// SIMATIC S7-200 project (STEP 7-Micro/WIN), CPU 226 REL 01.23

SYMBOL_TABLE USER1
start_button     I0.0     // start button
stop_button      I0.1     // stop button
inner_c_1_m      I0.2     // inner calling for first floor ( modern lift )
inner_c_2_m      I0.3     // inner calling for second floor ( modern lift )
inner_c_3_m      I0.4     // inner calling for third floor ( modern lift )
emergency_button I0.5     // system emergency button ( modern lift )
door_sensor_m    I0.6     // cabin door sensor ( modern lift )
bottom_limit_m   I0.7     // bottom limit sensor ( modern lift )
top_limit_m      I1.0     // top limit sensor ( modern lift )
floor_1_limit_m  I1.1     // first floor sensor ( modern lift )
floor_2_limit_m  I1.2     // second floor sensor ( modern lift )
floor_3_limit_m  I1.3     // third floor sensor ( modern lift )
floor_1_limit_o  I1.4     // first floor sensor ( old lift )
floor_2_limit_o  I1.5     // second floor sensor ( old lift )
floor_3_limit_o  I1.6     // third floor sensor ( old lift )
inner_c_1_o      I2.4     // inner calling for first floor ( old lift )
inner_c_2_o      I2.5     // inner calling for second floor ( old lift )
inner_c_3_o      I2.6     // inner calling for third floor ( old lift )
outer_c_1        I2.0     // outer calling for first floor
outer_c_2_d      I2.1     // outer calling for second floor in purpose of moving down
outer_c_2_u      I2.2     // outer calling for second floor in purpose of moving up
outer_c_3        I2.3     // outer calling for third floor
data_a_m         Q0.0     // data  a  for  (7447 7_segment) circuit  ( modern lift )
data_b_m         Q0.1     // data  b  for  (7447 7_segment) circuit  ( modern lift )
floor_1_led_m    Q0.2     // first floor calling led  ( modern lift )
floor_2_led_m    Q0.3     // second floor calling led  ( modern lift )
floor_3_led_m    Q0.4     // third floor calling led  ( modern lift )
emergency_led    Q0.5     // emergency calling led  ( modern lift )
door_lock_m      Q0.6     // security lock open/close output for lift cabin door  ( modern lift )
lighting_m       Q0.7     // cabin  inside lighting  ( modern lift )
cabin_down_m     Q1.0     // output for the lift motor for down movement  ( modern lift )
cabin_up_m       Q1.1     // output for the lift motor for up movement  ( modern lift )
cabin_down_o     Q1.3     // output for the lift motor for down movement  ( old lift )
cabin_up_o       Q1.2     // output for the lift motor for up movement  ( old lift )
functional_timer_off_1 T37      // functional_timer_off is used specially for inside cabin lighting
functional_timer_off_2 T38      // functional_timer_off is used in purpose of delaying between calls (modern lift)
functional_timer_off_3 T39      // functional_timer_off is used in purpose of delaying between calls (old lift)
functional_byte_1 VB0      // functional_byte_is used to determine in which floor is modern lift
functional_byte_2 VB1      // functional_byte_is used to determine in which floor is old lif
functional_bit_0 V6.0     // bit used for downloading the starting constraints in sbr(1) and sbr(2)
functional_bit_1 V6.1     // bit used for downloading the starting constraints in sbr(3)
functional_bit_2 V6.2     // bit used for downloading the starting constraints in sbr(4)
functional_bit_3 V6.3     // bit used for downloading the starting constraints in sbr(5)
functional_bit_4 V6.4     // bit used for downloading the starting constraints in sbr(6)
functional_bit_5 V6.5     // bit used for downloading the starting constraints in sbr(7)
functional_bit_6 V6.6     // bit used for downloading the starting constraints in sbr(11)
functional_bit_7 V6.7     // bit used for downloading the starting constraints in sbr(12)
functional_bit_8 V7.0     // bit used for downloading the starting constraints in sbr(13)
functional_bit_9 V7.1     // bit used for downloading the starting constraints in sbr(14)
system_on_off    M0.0     // system  on/off contact
sbr_1_call_bit   M0.1     // subroutine (1) calling bit
sbr_2_call_bit   M0.2     // subroutine (2) calling bit
sbr_3_call_bit   M0.3     // subroutine (3) calling bit
sbr_4_call_bit   M0.4     // subroutine (4) calling bit
sbr_5_call_bit   M0.5     // subroutine (5) calling bit
sbr_6_call_bit   M0.6     // subroutine (6) calling bit
sbr_7_call_bit   M0.7     // subroutine (7) calling bit
sbr_11_call_bit  M2.3     // subroutine (11) calling bit
sbr_12_call_bit  M2.7     // subroutine (12) calling bit
sbr_13_call_bit  M3.0     // subroutine (13) calling bit
sbr_14_call_bit  M3.1     // subroutine (14) calling bit
m_1_to_2         M1.0     // it is made set while modern lift is moving from floor 1 to floor 2
m_2_to_3         M1.1     // it is made set while modern lift is moving from floor 2 to floor 3
m_2_to_1         M1.2     // it is made set while modern lift is moving from floor 2 to floor 1
m_3_to_2         M1.3     // it is made set while modern lift is moving from floor 3 to floor 2
m_busy           M1.4     // it is made set while modern lift is busy
o_1_to_2         M1.5     // it is made set while old lift is moving from floor 1 to floor 2
o_2_to_3         M1.6     // it is made set while old lift is moving from floor 2 to floor 3
o_2_to_1         M1.7     // it is made set while old lift is moving from floor 2 to floor 1
o_3_to_2         M2.0     // it is made set while old lift is moving from floor 3 to floor 2
o_busy           M2.1     // it is made set while old lift is busy
both_ready       M2.2     // it is made set when both lifts are ready
m_busy_o_ready   M2.4     // it is made set when modren lift is busy and old lift is ready
m_ready_o_busy   M2.5     // it is made set when modren lift is ready and old lift is busy
both_busy        M2.6     // it is made set when both lifts are busy
First_Scan_On    SM0.1    // ON for the first scan cycle only
Always_On        SM0.0    // Always ON
END_SYMBOL_TABLE

ORGANIZATION_BLOCK MAIN:OB1
TITLE=control two lifts (modern and old) to work in priority
BEGIN
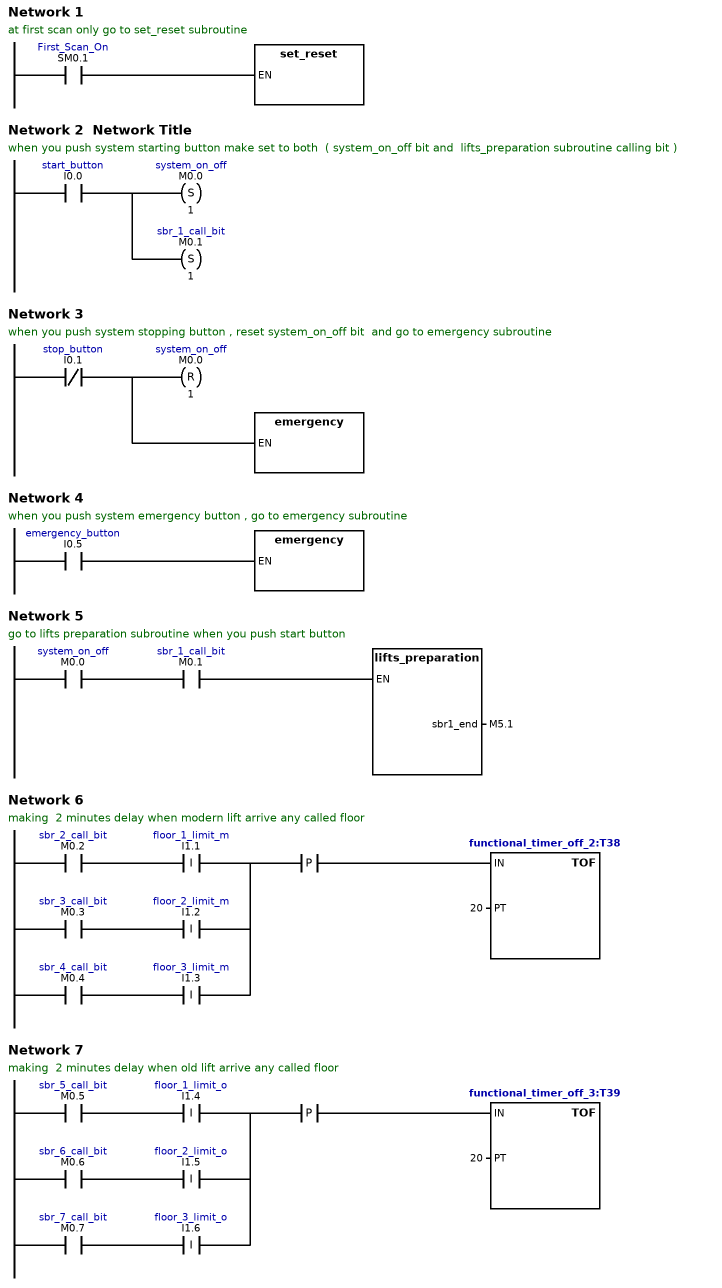
Network 1
// at first scan only go to set_reset subroutine
LD     First_Scan_On:SM0.1
CALL   set_reset:SBR0
Network 2 // Network Title
// when you push system starting button make set to both  ( system_on_off bit and  lifts_preparation subroutine calling bit )
LD     start_button:I0.0
S      system_on_off:M0.0, 1
S      sbr_1_call_bit:M0.1, 1
Network 3
// when you push system stopping button , reset system_on_off bit  and go to emergency subroutine
LDN    stop_button:I0.1
R      system_on_off:M0.0, 1
CALL   emergency:SBR15
Network 4
// when you push system emergency button , go to emergency subroutine
LD     emergency_button:I0.5
CALL   emergency:SBR15
Network 5
// go to lifts preparation subroutine when you push start button
LD     system_on_off:M0.0
A      sbr_1_call_bit:M0.1
CALL   lifts_preparation:SBR1, M5.1
Network 6
// making  2 minutes delay when modern lift arrive any called floor
LD     sbr_2_call_bit:M0.2
AI     floor_1_limit_m:I1.1
LD     sbr_3_call_bit:M0.3
AI     floor_2_limit_m:I1.2
OLD
LD     sbr_4_call_bit:M0.4
AI     floor_3_limit_m:I1.3
OLD
EU
TOF    functional_timer_off_2:T38, 20
Network 7
// making  2 minutes delay when old lift arrive any called floor
LD     sbr_5_call_bit:M0.5
AI     floor_1_limit_o:I1.4
LD     sbr_6_call_bit:M0.6
AI     floor_2_limit_o:I1.5
OLD
LD     sbr_7_call_bit:M0.7
AI     floor_3_limit_o:I1.6
OLD
EU
TOF    functional_timer_off_3:T39, 20
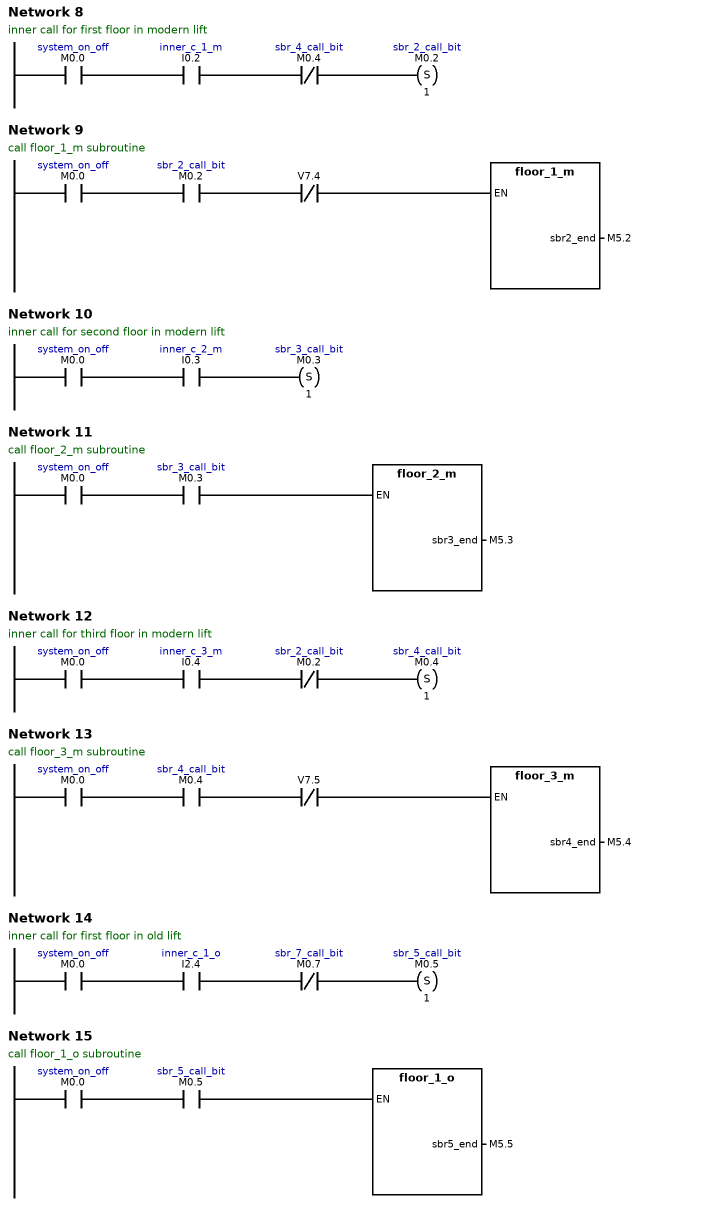
Network 8
// inner call for first floor in modern lift
LD     system_on_off:M0.0
A      inner_c_1_m:I0.2
AN     sbr_4_call_bit:M0.4
S      sbr_2_call_bit:M0.2, 1
Network 9
// call floor_1_m subroutine
LD     system_on_off:M0.0
A      sbr_2_call_bit:M0.2
AN     V7.4
CALL   floor_1_m:SBR2, M5.2
Network 10
// inner call for second floor in modern lift
LD     system_on_off:M0.0
A      inner_c_2_m:I0.3
S      sbr_3_call_bit:M0.3, 1
Network 11
// call floor_2_m subroutine
LD     system_on_off:M0.0
A      sbr_3_call_bit:M0.3
CALL   floor_2_m:SBR3, M5.3
Network 12
// inner call for third floor in modern lift
LD     system_on_off:M0.0
A      inner_c_3_m:I0.4
AN     sbr_2_call_bit:M0.2
S      sbr_4_call_bit:M0.4, 1
Network 13
// call floor_3_m subroutine
LD     system_on_off:M0.0
A      sbr_4_call_bit:M0.4
AN     V7.5
CALL   floor_3_m:SBR4, M5.4
Network 14
// inner call for first floor in old lift
LD     system_on_off:M0.0
A      inner_c_1_o:I2.4
AN     sbr_7_call_bit:M0.7
S      sbr_5_call_bit:M0.5, 1
Network 15
// call floor_1_o subroutine
LD     system_on_off:M0.0
A      sbr_5_call_bit:M0.5
CALL   floor_1_o:SBR5, M5.5
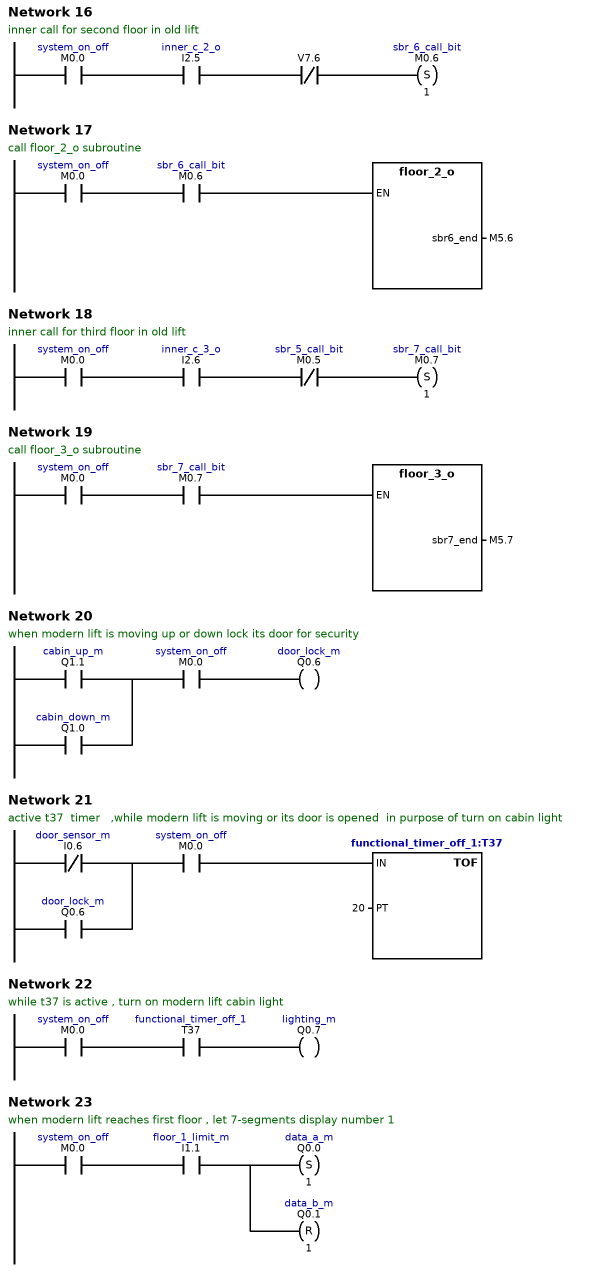
Network 16
// inner call for second floor in old lift
LD     system_on_off:M0.0
A      inner_c_2_o:I2.5
AN     V7.6
S      sbr_6_call_bit:M0.6, 1
Network 17
// call floor_2_o subroutine
LD     system_on_off:M0.0
A      sbr_6_call_bit:M0.6
CALL   floor_2_o:SBR6, M5.6
Network 18
// inner call for third floor in old lift
LD     system_on_off:M0.0
A      inner_c_3_o:I2.6
AN     sbr_5_call_bit:M0.5
S      sbr_7_call_bit:M0.7, 1
Network 19
// call floor_3_o subroutine
LD     system_on_off:M0.0
A      sbr_7_call_bit:M0.7
CALL   floor_3_o:SBR7, M5.7
Network 20
// when modern lift is moving up or down lock its door for security
LD     cabin_up_m:Q1.1
O      cabin_down_m:Q1.0
A      system_on_off:M0.0
=      door_lock_m:Q0.6
Network 21
// active t37  timer   ,while modern lift is moving or its door is opened  in purpose of turn on cabin light
LDN    door_sensor_m:I0.6
O      door_lock_m:Q0.6
A      system_on_off:M0.0
TOF    functional_timer_off_1:T37, 20
Network 22
// while t37 is active , turn on modern lift cabin light 
LD     system_on_off:M0.0
A      functional_timer_off_1:T37
=      lighting_m:Q0.7
Network 23
// when modern lift reaches first floor , let 7-segments display number 1
LD     system_on_off:M0.0
A      floor_1_limit_m:I1.1
S      data_a_m:Q0.0, 1
R      data_b_m:Q0.1, 1
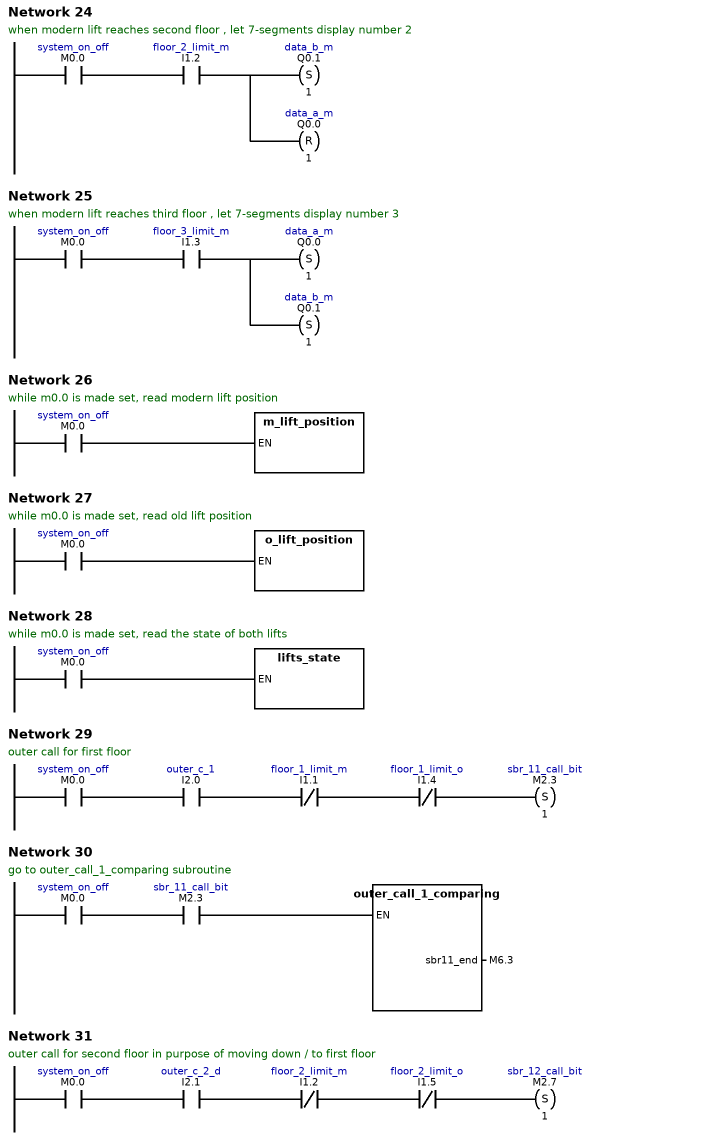
Network 24
// when modern lift reaches second floor , let 7-segments display number 2
LD     system_on_off:M0.0
A      floor_2_limit_m:I1.2
S      data_b_m:Q0.1, 1
R      data_a_m:Q0.0, 1
Network 25
// when modern lift reaches third floor , let 7-segments display number 3
LD     system_on_off:M0.0
A      floor_3_limit_m:I1.3
S      data_a_m:Q0.0, 1
S      data_b_m:Q0.1, 1
Network 26
// while m0.0 is made set, read modern lift position
LD     system_on_off:M0.0
CALL   m_lift_position:SBR8
Network 27
// while m0.0 is made set, read old lift position
LD     system_on_off:M0.0
CALL   o_lift_position:SBR9
Network 28
// while m0.0 is made set, read the state of both lifts
LD     system_on_off:M0.0
CALL   lifts_state:SBR10
Network 29
// outer call for first floor  
LD     system_on_off:M0.0
A      outer_c_1:I2.0
AN     floor_1_limit_m:I1.1
AN     floor_1_limit_o:I1.4
S      sbr_11_call_bit:M2.3, 1
Network 30
// go to outer_call_1_comparing subroutine
LD     system_on_off:M0.0
A      sbr_11_call_bit:M2.3
CALL   outer_call_1_comparing:SBR11, M6.3
Network 31
// outer call for second floor in purpose of moving down / to first floor
LD     system_on_off:M0.0
A      outer_c_2_d:I2.1
AN     floor_2_limit_m:I1.2
AN     floor_2_limit_o:I1.5
S      sbr_12_call_bit:M2.7, 1
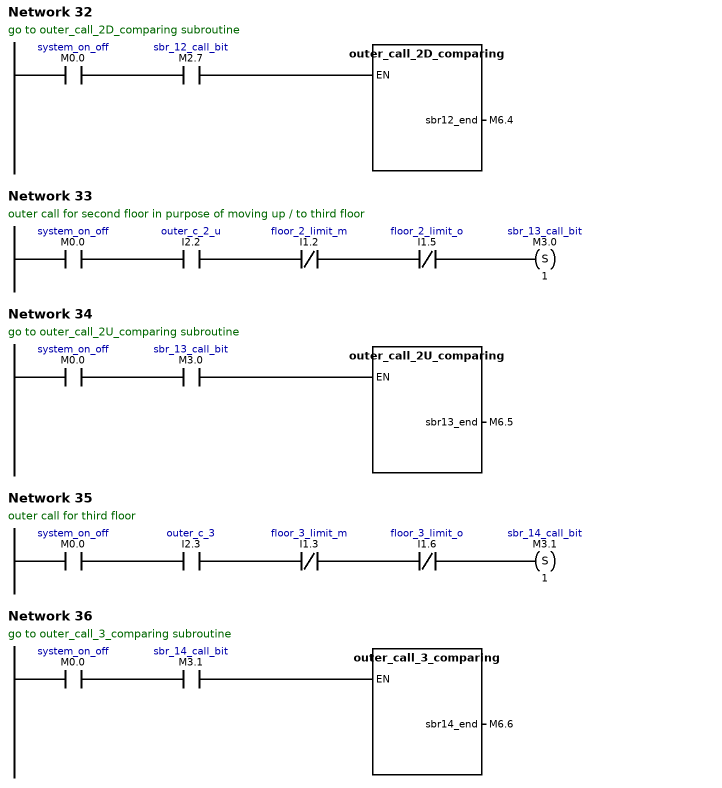
Network 32
// go to outer_call_2D_comparing subroutine
LD     system_on_off:M0.0
A      sbr_12_call_bit:M2.7
CALL   outer_call_2D_comparing:SBR12, M6.4
Network 33
// outer call for second floor in purpose of moving up / to third floor
LD     system_on_off:M0.0
A      outer_c_2_u:I2.2
AN     floor_2_limit_m:I1.2
AN     floor_2_limit_o:I1.5
S      sbr_13_call_bit:M3.0, 1
Network 34
// go to outer_call_2U_comparing subroutine
LD     system_on_off:M0.0
A      sbr_13_call_bit:M3.0
CALL   outer_call_2U_comparing:SBR13, M6.5
Network 35
// outer call for third floor 
LD     system_on_off:M0.0
A      outer_c_3:I2.3
AN     floor_3_limit_m:I1.3
AN     floor_3_limit_o:I1.6
S      sbr_14_call_bit:M3.1, 1
Network 36
// go to outer_call_3_comparing subroutine
LD     system_on_off:M0.0
A      sbr_14_call_bit:M3.1
CALL   outer_call_3_comparing:SBR14, M6.6
END_ORGANIZATION_BLOCK

SUBROUTINE_BLOCK set_reset:SBR0
TITLE=put all memories , timers and outputs that are used in program at initial position 
BEGIN
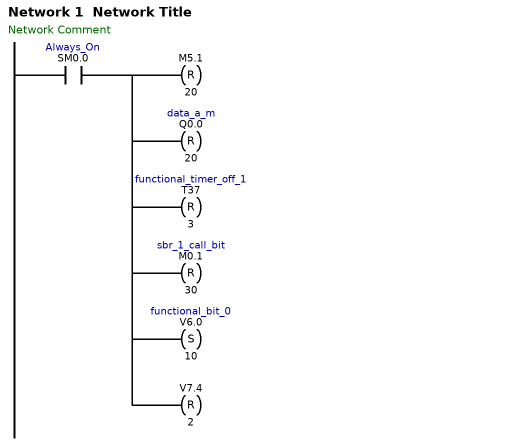
Network 1 // Network Title
// Network Comment
LD     Always_On:SM0.0
R      M5.1, 20
R      data_a_m:Q0.0, 20
R      functional_timer_off_1:T37, 3
R      sbr_1_call_bit:M0.1, 30
S      functional_bit_0:V6.0, 10
R      V7.4, 2
END_SUBROUTINE_BLOCK

SUBROUTINE_BLOCK lifts_preparation:SBR1
TITLE=move modern lift to third floor and old lift to first floor 
VAR_OUTPUT
sbr1_end:BOOL;	// L0.0 
END_VAR
BEGIN
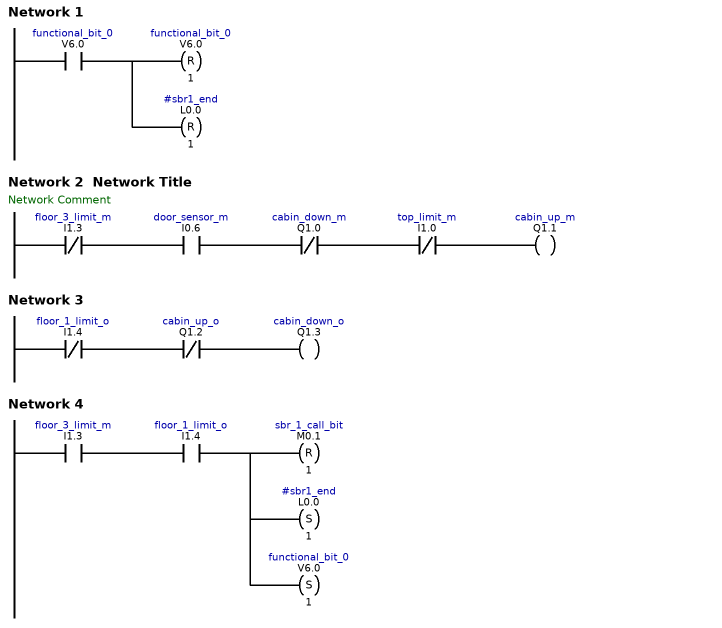
Network 1
LD     functional_bit_0:V6.0
R      functional_bit_0:V6.0, 1
R      #sbr1_end:L0.0, 1
Network 2 // Network Title
// Network Comment
LDN    floor_3_limit_m:I1.3
A      door_sensor_m:I0.6
AN     cabin_down_m:Q1.0
AN     top_limit_m:I1.0
=      cabin_up_m:Q1.1
Network 3
LDN    floor_1_limit_o:I1.4
AN     cabin_up_o:Q1.2
=      cabin_down_o:Q1.3
Network 4
LD     floor_3_limit_m:I1.3
A      floor_1_limit_o:I1.4
R      sbr_1_call_bit:M0.1, 1
S      #sbr1_end:L0.0, 1
S      functional_bit_0:V6.0, 1
END_SUBROUTINE_BLOCK

SUBROUTINE_BLOCK floor_1_m:SBR2
TITLE=move modern lift to first floor
VAR_OUTPUT
sbr2_end:BOOL;	// L0.0 
END_VAR
BEGIN
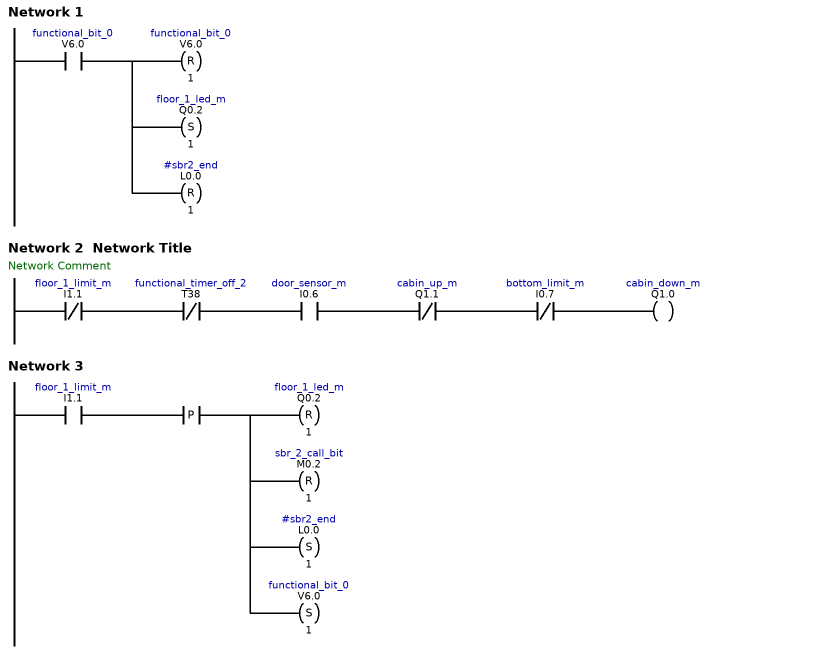
Network 1
LD     functional_bit_0:V6.0
R      functional_bit_0:V6.0, 1
S      floor_1_led_m:Q0.2, 1
R      #sbr2_end:L0.0, 1
Network 2 // Network Title
// Network Comment
LDN    floor_1_limit_m:I1.1
AN     functional_timer_off_2:T38
A      door_sensor_m:I0.6
AN     cabin_up_m:Q1.1
AN     bottom_limit_m:I0.7
=      cabin_down_m:Q1.0
Network 3
LD     floor_1_limit_m:I1.1
EU
R      floor_1_led_m:Q0.2, 1
R      sbr_2_call_bit:M0.2, 1
S      #sbr2_end:L0.0, 1
S      functional_bit_0:V6.0, 1
END_SUBROUTINE_BLOCK

SUBROUTINE_BLOCK floor_2_m:SBR3
TITLE=move modern lift to second floor
VAR_OUTPUT
sbr3_end:BOOL;	// L0.0 
END_VAR
BEGIN
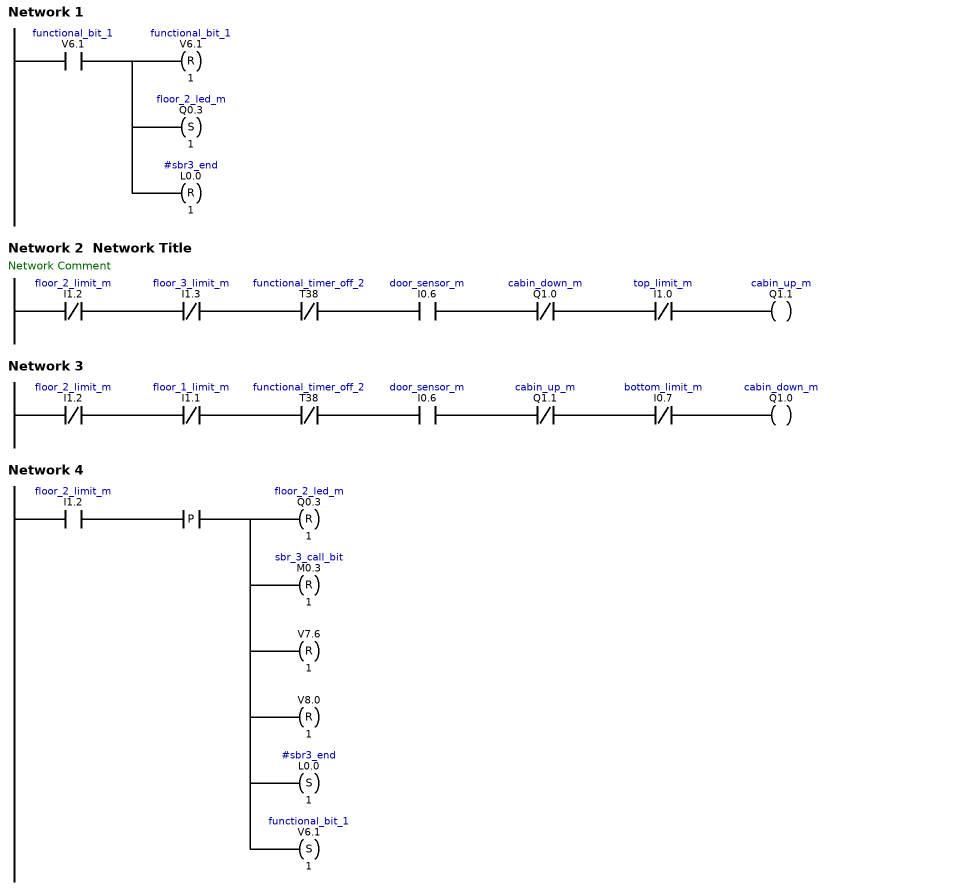
Network 1
LD     functional_bit_1:V6.1
R      functional_bit_1:V6.1, 1
S      floor_2_led_m:Q0.3, 1
R      #sbr3_end:L0.0, 1
Network 2 // Network Title
// Network Comment
LDN    floor_2_limit_m:I1.2
AN     floor_3_limit_m:I1.3
AN     functional_timer_off_2:T38
A      door_sensor_m:I0.6
AN     cabin_down_m:Q1.0
AN     top_limit_m:I1.0
=      cabin_up_m:Q1.1
Network 3
LDN    floor_2_limit_m:I1.2
AN     floor_1_limit_m:I1.1
AN     functional_timer_off_2:T38
A      door_sensor_m:I0.6
AN     cabin_up_m:Q1.1
AN     bottom_limit_m:I0.7
=      cabin_down_m:Q1.0
Network 4
LD     floor_2_limit_m:I1.2
EU
R      floor_2_led_m:Q0.3, 1
R      sbr_3_call_bit:M0.3, 1
R      V7.6, 1
R      V8.0, 1
S      #sbr3_end:L0.0, 1
S      functional_bit_1:V6.1, 1
END_SUBROUTINE_BLOCK

SUBROUTINE_BLOCK floor_3_m:SBR4
TITLE=move modern lift to third floor
VAR_OUTPUT
sbr4_end:BOOL;	// L0.0 
END_VAR
BEGIN
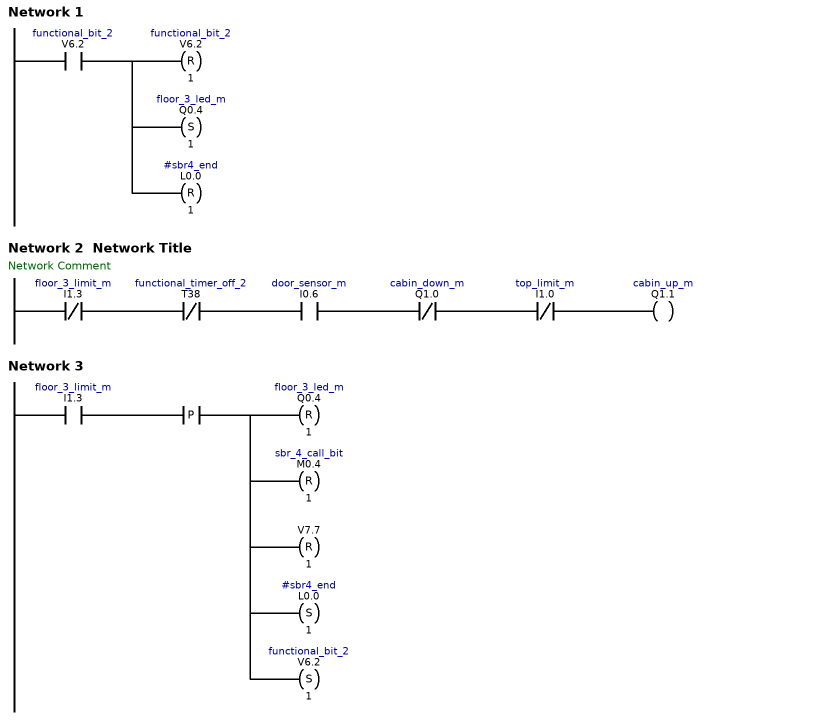
Network 1
LD     functional_bit_2:V6.2
R      functional_bit_2:V6.2, 1
S      floor_3_led_m:Q0.4, 1
R      #sbr4_end:L0.0, 1
Network 2 // Network Title
// Network Comment
LDN    floor_3_limit_m:I1.3
AN     functional_timer_off_2:T38
A      door_sensor_m:I0.6
AN     cabin_down_m:Q1.0
AN     top_limit_m:I1.0
=      cabin_up_m:Q1.1
Network 3
LD     floor_3_limit_m:I1.3
EU
R      floor_3_led_m:Q0.4, 1
R      sbr_4_call_bit:M0.4, 1
R      V7.7, 1
S      #sbr4_end:L0.0, 1
S      functional_bit_2:V6.2, 1
END_SUBROUTINE_BLOCK

SUBROUTINE_BLOCK floor_1_o:SBR5
TITLE=move old lift to first floor
VAR_OUTPUT
sbr5_end:BOOL;	// L0.0 
END_VAR
BEGIN
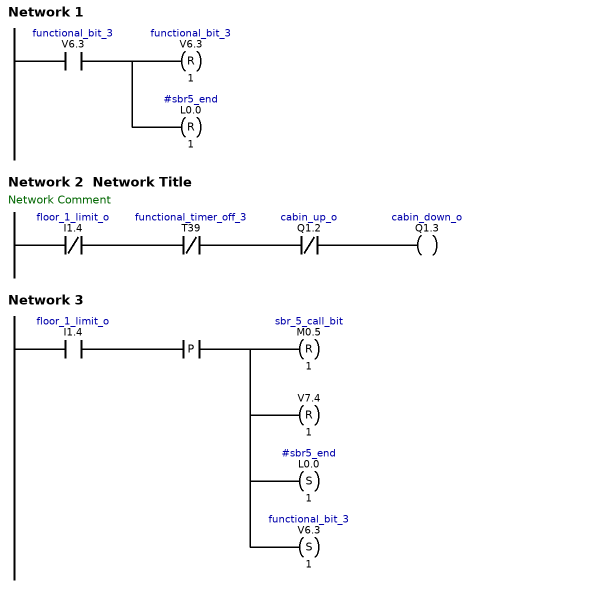
Network 1
LD     functional_bit_3:V6.3
R      functional_bit_3:V6.3, 1
R      #sbr5_end:L0.0, 1
Network 2 // Network Title
// Network Comment
LDN    floor_1_limit_o:I1.4
AN     functional_timer_off_3:T39
AN     cabin_up_o:Q1.2
=      cabin_down_o:Q1.3
Network 3
LD     floor_1_limit_o:I1.4
EU
R      sbr_5_call_bit:M0.5, 1
R      V7.4, 1
S      #sbr5_end:L0.0, 1
S      functional_bit_3:V6.3, 1
END_SUBROUTINE_BLOCK

SUBROUTINE_BLOCK floor_2_o:SBR6
TITLE=move old lift to second floor
VAR_OUTPUT
sbr6_end:BOOL;	// L0.0 
END_VAR
BEGIN
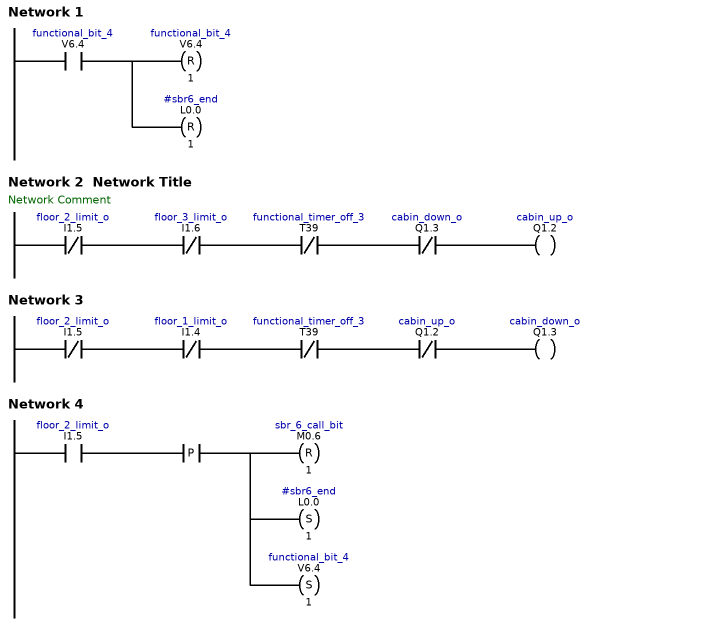
Network 1
LD     functional_bit_4:V6.4
R      functional_bit_4:V6.4, 1
R      #sbr6_end:L0.0, 1
Network 2 // Network Title
// Network Comment
LDN    floor_2_limit_o:I1.5
AN     floor_3_limit_o:I1.6
AN     functional_timer_off_3:T39
AN     cabin_down_o:Q1.3
=      cabin_up_o:Q1.2
Network 3
LDN    floor_2_limit_o:I1.5
AN     floor_1_limit_o:I1.4
AN     functional_timer_off_3:T39
AN     cabin_up_o:Q1.2
=      cabin_down_o:Q1.3
Network 4
LD     floor_2_limit_o:I1.5
EU
R      sbr_6_call_bit:M0.6, 1
S      #sbr6_end:L0.0, 1
S      functional_bit_4:V6.4, 1
END_SUBROUTINE_BLOCK

SUBROUTINE_BLOCK floor_3_o:SBR7
TITLE=move old lift to third floor
VAR_OUTPUT
sbr7_end:BOOL;	// L0.0 
END_VAR
BEGIN
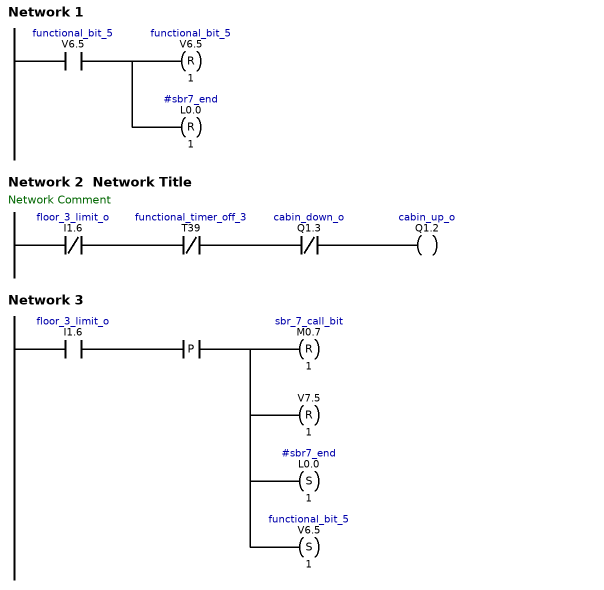
Network 1
LD     functional_bit_5:V6.5
R      functional_bit_5:V6.5, 1
R      #sbr7_end:L0.0, 1
Network 2 // Network Title
// Network Comment
LDN    floor_3_limit_o:I1.6
AN     functional_timer_off_3:T39
AN     cabin_down_o:Q1.3
=      cabin_up_o:Q1.2
Network 3
LD     floor_3_limit_o:I1.6
EU
R      sbr_7_call_bit:M0.7, 1
R      V7.5, 1
S      #sbr7_end:L0.0, 1
S      functional_bit_5:V6.5, 1
END_SUBROUTINE_BLOCK

SUBROUTINE_BLOCK m_lift_position:SBR8
TITLE=determine the position of modern lift (ex: moving form 1st floor to 2st floor )
BEGIN
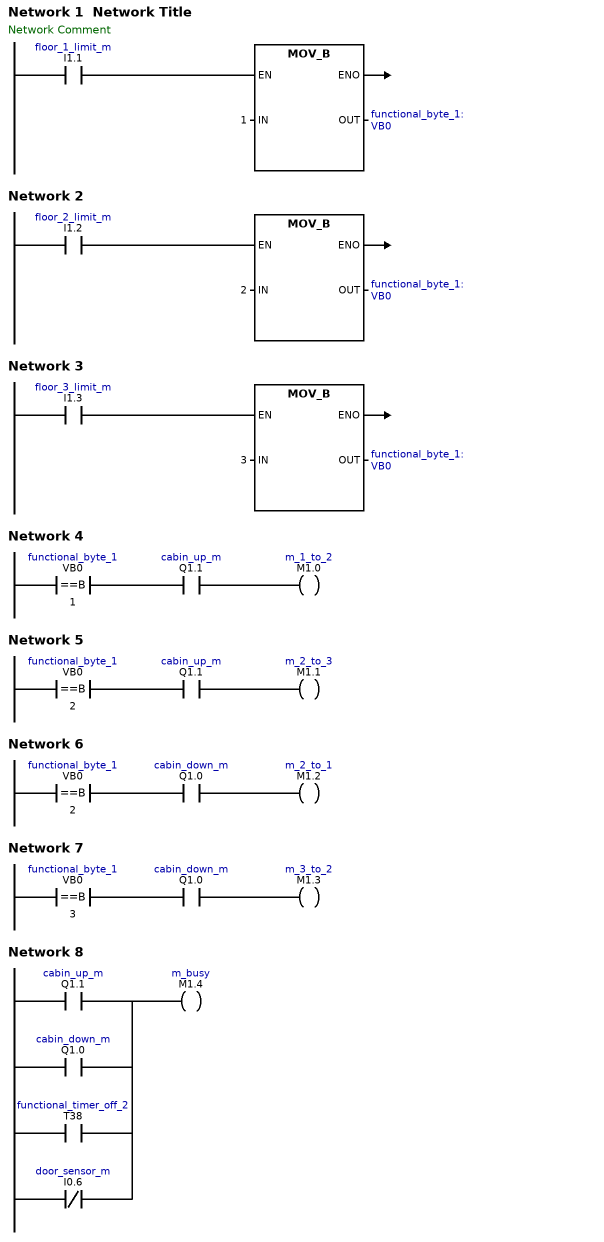
Network 1 // Network Title
// Network Comment
LD     floor_1_limit_m:I1.1
MOVB   1, functional_byte_1:VB0
Network 2
LD     floor_2_limit_m:I1.2
MOVB   2, functional_byte_1:VB0
Network 3
LD     floor_3_limit_m:I1.3
MOVB   3, functional_byte_1:VB0
Network 4
LDB=   functional_byte_1:VB0, 1
A      cabin_up_m:Q1.1
=      m_1_to_2:M1.0
Network 5
LDB=   functional_byte_1:VB0, 2
A      cabin_up_m:Q1.1
=      m_2_to_3:M1.1
Network 6
LDB=   functional_byte_1:VB0, 2
A      cabin_down_m:Q1.0
=      m_2_to_1:M1.2
Network 7
LDB=   functional_byte_1:VB0, 3
A      cabin_down_m:Q1.0
=      m_3_to_2:M1.3
Network 8
LD     cabin_up_m:Q1.1
O      cabin_down_m:Q1.0
O      functional_timer_off_2:T38
ON     door_sensor_m:I0.6
=      m_busy:M1.4
END_SUBROUTINE_BLOCK

SUBROUTINE_BLOCK o_lift_position:SBR9
TITLE=determine the position of old lift (ex: moving form 3st floor to 2st floor )
BEGIN
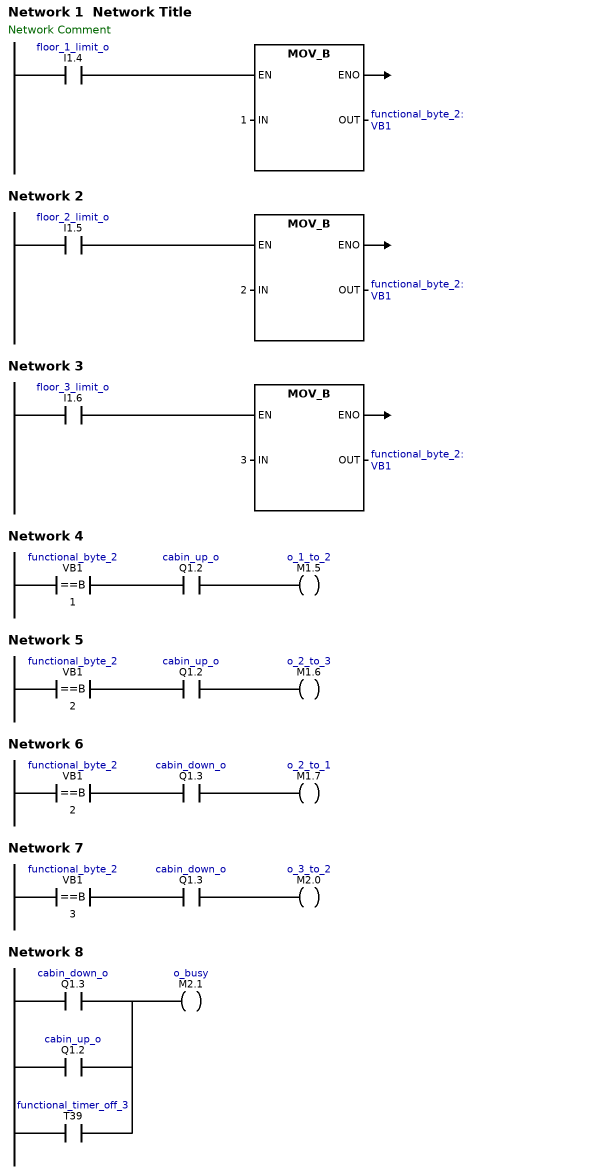
Network 1 // Network Title
// Network Comment
LD     floor_1_limit_o:I1.4
MOVB   1, functional_byte_2:VB1
Network 2
LD     floor_2_limit_o:I1.5
MOVB   2, functional_byte_2:VB1
Network 3
LD     floor_3_limit_o:I1.6
MOVB   3, functional_byte_2:VB1
Network 4
LDB=   functional_byte_2:VB1, 1
A      cabin_up_o:Q1.2
=      o_1_to_2:M1.5
Network 5
LDB=   functional_byte_2:VB1, 2
A      cabin_up_o:Q1.2
=      o_2_to_3:M1.6
Network 6
LDB=   functional_byte_2:VB1, 2
A      cabin_down_o:Q1.3
=      o_2_to_1:M1.7
Network 7
LDB=   functional_byte_2:VB1, 3
A      cabin_down_o:Q1.3
=      o_3_to_2:M2.0
Network 8
LD     cabin_down_o:Q1.3
O      cabin_up_o:Q1.2
O      functional_timer_off_3:T39
=      o_busy:M2.1
END_SUBROUTINE_BLOCK

SUBROUTINE_BLOCK lifts_state:SBR10
TITLE=determine the state of both lifts  (ex1: both are ready .  ex2:modern lift is busy and old is ready )
BEGIN
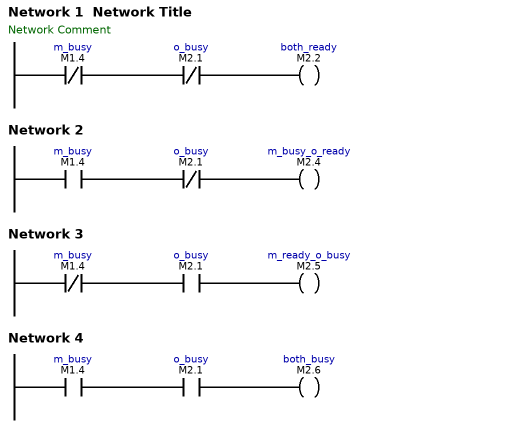
Network 1 // Network Title
// Network Comment
LDN    m_busy:M1.4
AN     o_busy:M2.1
=      both_ready:M2.2
Network 2
LD     m_busy:M1.4
AN     o_busy:M2.1
=      m_busy_o_ready:M2.4
Network 3
LDN    m_busy:M1.4
A      o_busy:M2.1
=      m_ready_o_busy:M2.5
Network 4
LD     m_busy:M1.4
A      o_busy:M2.1
=      both_busy:M2.6
END_SUBROUTINE_BLOCK

SUBROUTINE_BLOCK outer_call_1_comparing:SBR11
TITLE=outer call from first floor .
// according to ( modern position , old position and lifts state ) , do logical comparison  to determine which lift will move to first floor
VAR_OUTPUT
sbr11_end:BOOL;	// L0.0 
END_VAR
BEGIN
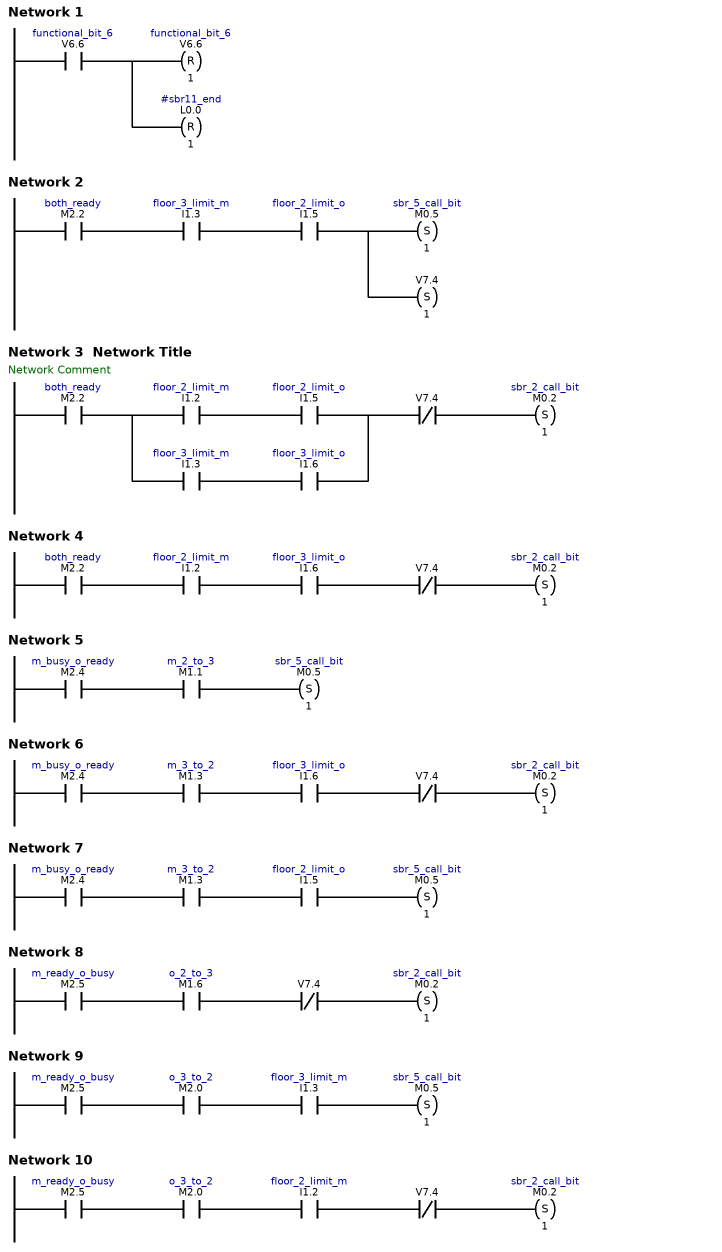
Network 1
LD     functional_bit_6:V6.6
R      functional_bit_6:V6.6, 1
R      #sbr11_end:L0.0, 1
Network 2
LD     both_ready:M2.2
A      floor_3_limit_m:I1.3
A      floor_2_limit_o:I1.5
S      sbr_5_call_bit:M0.5, 1
S      V7.4, 1
Network 3 // Network Title
// Network Comment
LD     both_ready:M2.2
LD     floor_2_limit_m:I1.2
A      floor_2_limit_o:I1.5
LD     floor_3_limit_m:I1.3
A      floor_3_limit_o:I1.6
OLD
ALD
AN     V7.4
S      sbr_2_call_bit:M0.2, 1
Network 4
LD     both_ready:M2.2
A      floor_2_limit_m:I1.2
A      floor_3_limit_o:I1.6
AN     V7.4
S      sbr_2_call_bit:M0.2, 1
Network 5
LD     m_busy_o_ready:M2.4
A      m_2_to_3:M1.1
S      sbr_5_call_bit:M0.5, 1
Network 6
LD     m_busy_o_ready:M2.4
A      m_3_to_2:M1.3
A      floor_3_limit_o:I1.6
AN     V7.4
S      sbr_2_call_bit:M0.2, 1
Network 7
LD     m_busy_o_ready:M2.4
A      m_3_to_2:M1.3
A      floor_2_limit_o:I1.5
S      sbr_5_call_bit:M0.5, 1
Network 8
LD     m_ready_o_busy:M2.5
A      o_2_to_3:M1.6
AN     V7.4
S      sbr_2_call_bit:M0.2, 1
Network 9
LD     m_ready_o_busy:M2.5
A      o_3_to_2:M2.0
A      floor_3_limit_m:I1.3
S      sbr_5_call_bit:M0.5, 1
Network 10
LD     m_ready_o_busy:M2.5
A      o_3_to_2:M2.0
A      floor_2_limit_m:I1.2
AN     V7.4
S      sbr_2_call_bit:M0.2, 1
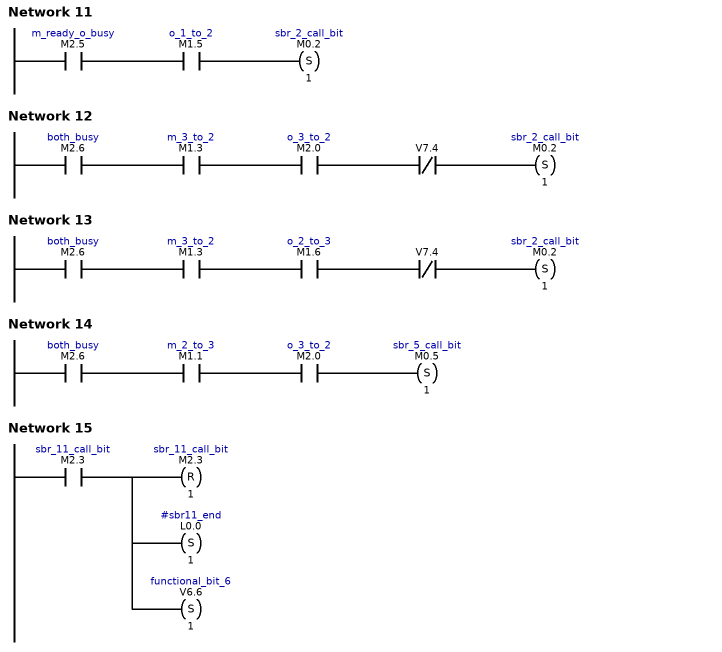
Network 11
LD     m_ready_o_busy:M2.5
A      o_1_to_2:M1.5
S      sbr_2_call_bit:M0.2, 1
Network 12
LD     both_busy:M2.6
A      m_3_to_2:M1.3
A      o_3_to_2:M2.0
AN     V7.4
S      sbr_2_call_bit:M0.2, 1
Network 13
LD     both_busy:M2.6
A      m_3_to_2:M1.3
A      o_2_to_3:M1.6
AN     V7.4
S      sbr_2_call_bit:M0.2, 1
Network 14
LD     both_busy:M2.6
A      m_2_to_3:M1.1
A      o_3_to_2:M2.0
S      sbr_5_call_bit:M0.5, 1
Network 15
LD     sbr_11_call_bit:M2.3
R      sbr_11_call_bit:M2.3, 1
S      #sbr11_end:L0.0, 1
S      functional_bit_6:V6.6, 1
END_SUBROUTINE_BLOCK

SUBROUTINE_BLOCK outer_call_2D_comparing:SBR12
TITLE=outer call from second floor in purpose of moving down to first floor . 
// according to ( modern position , old position and lifts state ) , do logical comparison  to determine which lift will move to second floor .
VAR_OUTPUT
sbr12_end:BOOL;	// L0.0 
END_VAR
BEGIN
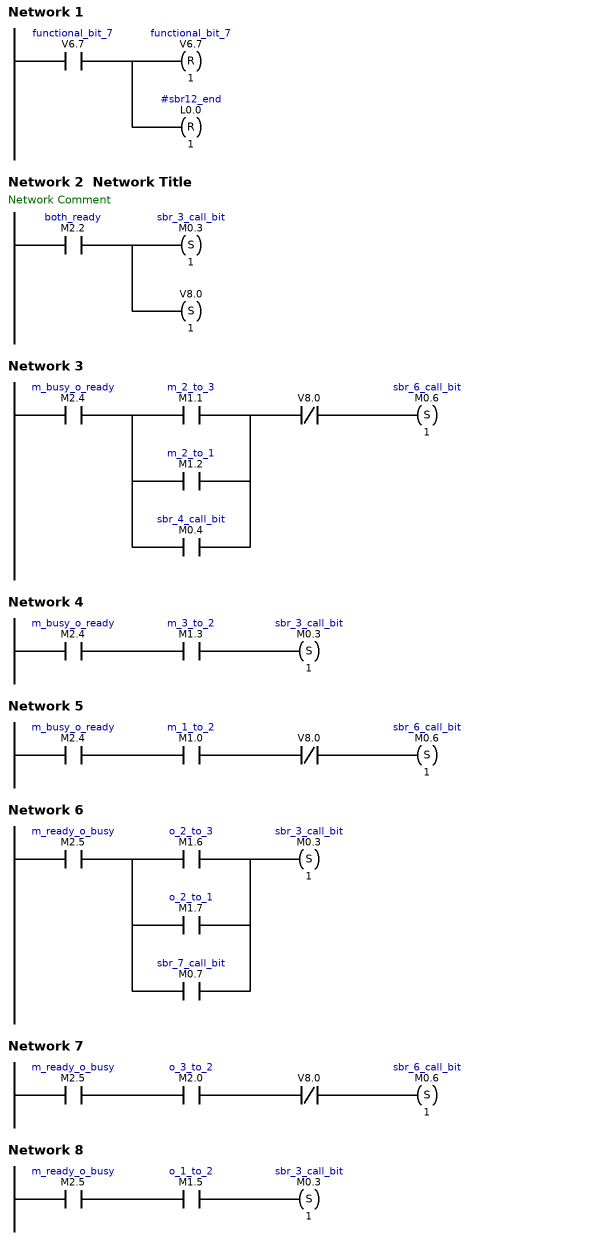
Network 1
LD     functional_bit_7:V6.7
R      functional_bit_7:V6.7, 1
R      #sbr12_end:L0.0, 1
Network 2 // Network Title
// Network Comment
LD     both_ready:M2.2
S      sbr_3_call_bit:M0.3, 1
S      V8.0, 1
Network 3
LD     m_busy_o_ready:M2.4
LD     m_2_to_3:M1.1
O      m_2_to_1:M1.2
O      sbr_4_call_bit:M0.4
ALD
AN     V8.0
S      sbr_6_call_bit:M0.6, 1
Network 4
LD     m_busy_o_ready:M2.4
A      m_3_to_2:M1.3
S      sbr_3_call_bit:M0.3, 1
Network 5
LD     m_busy_o_ready:M2.4
A      m_1_to_2:M1.0
AN     V8.0
S      sbr_6_call_bit:M0.6, 1
Network 6
LD     m_ready_o_busy:M2.5
LD     o_2_to_3:M1.6
O      o_2_to_1:M1.7
O      sbr_7_call_bit:M0.7
ALD
S      sbr_3_call_bit:M0.3, 1
Network 7
LD     m_ready_o_busy:M2.5
A      o_3_to_2:M2.0
AN     V8.0
S      sbr_6_call_bit:M0.6, 1
Network 8
LD     m_ready_o_busy:M2.5
A      o_1_to_2:M1.5
S      sbr_3_call_bit:M0.3, 1
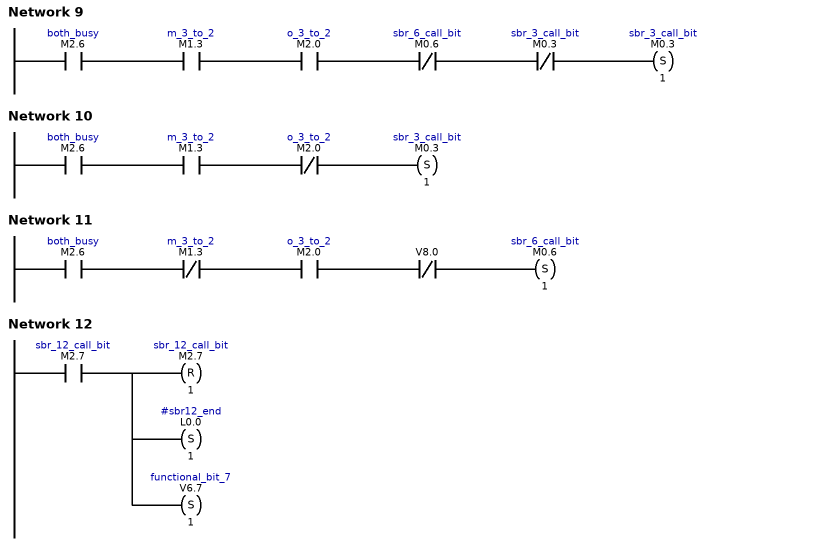
Network 9
LD     both_busy:M2.6
A      m_3_to_2:M1.3
A      o_3_to_2:M2.0
AN     sbr_6_call_bit:M0.6
AN     sbr_3_call_bit:M0.3
S      sbr_3_call_bit:M0.3, 1
Network 10
LD     both_busy:M2.6
A      m_3_to_2:M1.3
AN     o_3_to_2:M2.0
S      sbr_3_call_bit:M0.3, 1
Network 11
LD     both_busy:M2.6
AN     m_3_to_2:M1.3
A      o_3_to_2:M2.0
AN     V8.0
S      sbr_6_call_bit:M0.6, 1
Network 12
LD     sbr_12_call_bit:M2.7
R      sbr_12_call_bit:M2.7, 1
S      #sbr12_end:L0.0, 1
S      functional_bit_7:V6.7, 1
END_SUBROUTINE_BLOCK

SUBROUTINE_BLOCK outer_call_2U_comparing:SBR13
TITLE=outer call from second floor  in purpose of moving up to third floor .
// according to ( modern position , old position and lifts state ) , do logical comparison  to determine which lift will move to second floor .
VAR_OUTPUT
sbr13_end:BOOL;	// L0.0 
END_VAR
BEGIN
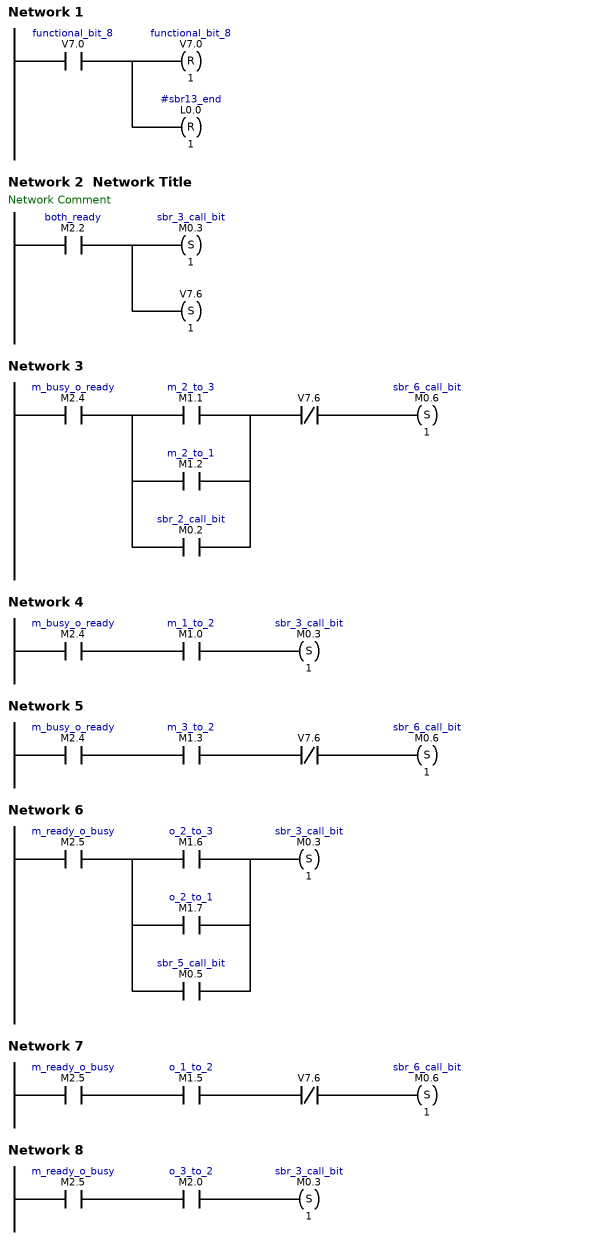
Network 1
LD     functional_bit_8:V7.0
R      functional_bit_8:V7.0, 1
R      #sbr13_end:L0.0, 1
Network 2 // Network Title
// Network Comment
LD     both_ready:M2.2
S      sbr_3_call_bit:M0.3, 1
S      V7.6, 1
Network 3
LD     m_busy_o_ready:M2.4
LD     m_2_to_3:M1.1
O      m_2_to_1:M1.2
O      sbr_2_call_bit:M0.2
ALD
AN     V7.6
S      sbr_6_call_bit:M0.6, 1
Network 4
LD     m_busy_o_ready:M2.4
A      m_1_to_2:M1.0
S      sbr_3_call_bit:M0.3, 1
Network 5
LD     m_busy_o_ready:M2.4
A      m_3_to_2:M1.3
AN     V7.6
S      sbr_6_call_bit:M0.6, 1
Network 6
LD     m_ready_o_busy:M2.5
LD     o_2_to_3:M1.6
O      o_2_to_1:M1.7
O      sbr_5_call_bit:M0.5
ALD
S      sbr_3_call_bit:M0.3, 1
Network 7
LD     m_ready_o_busy:M2.5
A      o_1_to_2:M1.5
AN     V7.6
S      sbr_6_call_bit:M0.6, 1
Network 8
LD     m_ready_o_busy:M2.5
A      o_3_to_2:M2.0
S      sbr_3_call_bit:M0.3, 1
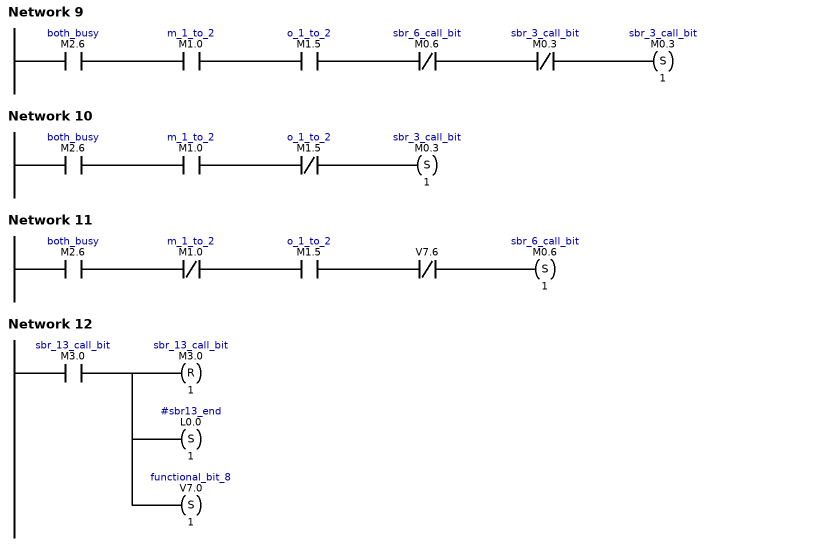
Network 9
LD     both_busy:M2.6
A      m_1_to_2:M1.0
A      o_1_to_2:M1.5
AN     sbr_6_call_bit:M0.6
AN     sbr_3_call_bit:M0.3
S      sbr_3_call_bit:M0.3, 1
Network 10
LD     both_busy:M2.6
A      m_1_to_2:M1.0
AN     o_1_to_2:M1.5
S      sbr_3_call_bit:M0.3, 1
Network 11
LD     both_busy:M2.6
AN     m_1_to_2:M1.0
A      o_1_to_2:M1.5
AN     V7.6
S      sbr_6_call_bit:M0.6, 1
Network 12
LD     sbr_13_call_bit:M3.0
R      sbr_13_call_bit:M3.0, 1
S      #sbr13_end:L0.0, 1
S      functional_bit_8:V7.0, 1
END_SUBROUTINE_BLOCK

SUBROUTINE_BLOCK outer_call_3_comparing:SBR14
TITLE=outer call from third floor .
// according to ( modern position , old position and lifts state ) , do logical comparison  to determine which lift will move to third floor
VAR_OUTPUT
sbr14_end:BOOL;	// L0.0 
END_VAR
BEGIN
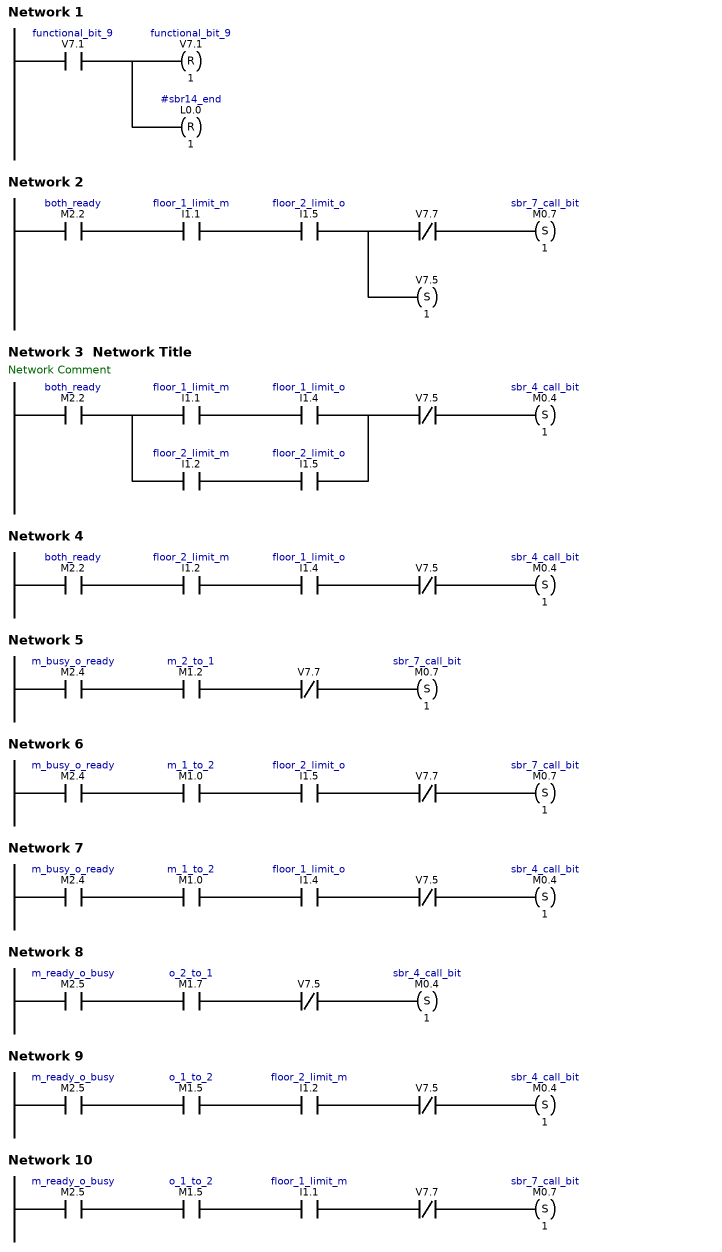
Network 1
LD     functional_bit_9:V7.1
R      functional_bit_9:V7.1, 1
R      #sbr14_end:L0.0, 1
Network 2
LD     both_ready:M2.2
A      floor_1_limit_m:I1.1
A      floor_2_limit_o:I1.5
LPS
AN     V7.7
S      sbr_7_call_bit:M0.7, 1
LPP
S      V7.5, 1
Network 3 // Network Title
// Network Comment
LD     both_ready:M2.2
LD     floor_1_limit_m:I1.1
A      floor_1_limit_o:I1.4
LD     floor_2_limit_m:I1.2
A      floor_2_limit_o:I1.5
OLD
ALD
AN     V7.5
S      sbr_4_call_bit:M0.4, 1
Network 4
LD     both_ready:M2.2
A      floor_2_limit_m:I1.2
A      floor_1_limit_o:I1.4
AN     V7.5
S      sbr_4_call_bit:M0.4, 1
Network 5
LD     m_busy_o_ready:M2.4
A      m_2_to_1:M1.2
AN     V7.7
S      sbr_7_call_bit:M0.7, 1
Network 6
LD     m_busy_o_ready:M2.4
A      m_1_to_2:M1.0
A      floor_2_limit_o:I1.5
AN     V7.7
S      sbr_7_call_bit:M0.7, 1
Network 7
LD     m_busy_o_ready:M2.4
A      m_1_to_2:M1.0
A      floor_1_limit_o:I1.4
AN     V7.5
S      sbr_4_call_bit:M0.4, 1
Network 8
LD     m_ready_o_busy:M2.5
A      o_2_to_1:M1.7
AN     V7.5
S      sbr_4_call_bit:M0.4, 1
Network 9
LD     m_ready_o_busy:M2.5
A      o_1_to_2:M1.5
A      floor_2_limit_m:I1.2
AN     V7.5
S      sbr_4_call_bit:M0.4, 1
Network 10
LD     m_ready_o_busy:M2.5
A      o_1_to_2:M1.5
A      floor_1_limit_m:I1.1
AN     V7.7
S      sbr_7_call_bit:M0.7, 1
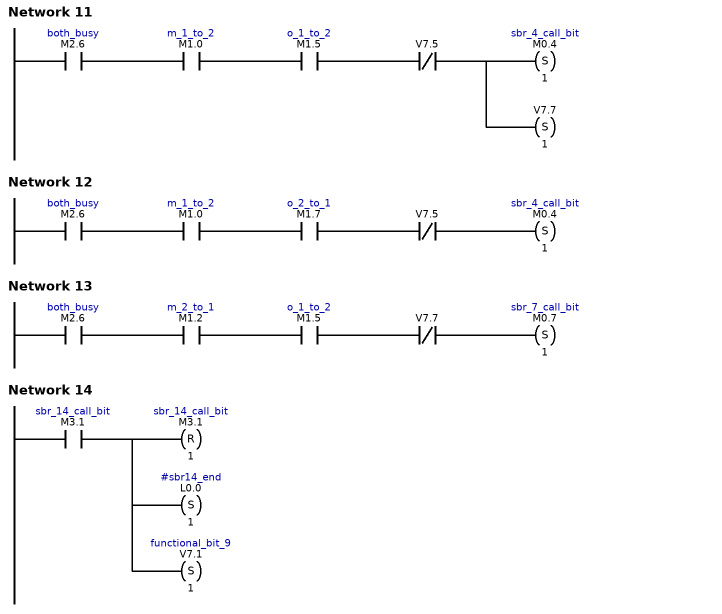
Network 11
LD     both_busy:M2.6
A      m_1_to_2:M1.0
A      o_1_to_2:M1.5
AN     V7.5
S      sbr_4_call_bit:M0.4, 1
S      V7.7, 1
Network 12
LD     both_busy:M2.6
A      m_1_to_2:M1.0
A      o_2_to_1:M1.7
AN     V7.5
S      sbr_4_call_bit:M0.4, 1
Network 13
LD     both_busy:M2.6
A      m_2_to_1:M1.2
A      o_1_to_2:M1.5
AN     V7.7
S      sbr_7_call_bit:M0.7, 1
Network 14
LD     sbr_14_call_bit:M3.1
R      sbr_14_call_bit:M3.1, 1
S      #sbr14_end:L0.0, 1
S      functional_bit_9:V7.1, 1
END_SUBROUTINE_BLOCK

SUBROUTINE_BLOCK emergency:SBR15
TITLE=reset ( memories, timers and outputs) that are used in the program ,and turn on emergency led .
BEGIN
